Fanuc KAREL source: kt00264.KL

-- PROVISIONAL review KL for V770-1; original PC SHA256 e8cb45a23f48b17e567031bccddfba465cc350efa91dea444729adb3129dde7d
-- Incomplete behavior may be omitted. Consult companion uncertainty JSON. Do not deploy.
PROGRAM KT00264
%NOLOCKGROUP
VAR
  R1 : REAL
  OUT : BOOLEAN
-- UNRESOLVED_DECL H2 type=002017
BEGIN
  -- UNRESOLVED_PC offsets 5-16; opcodes 2E,23
  -- UNRESOLVED_PC offsets 21-35; opcodes 2E,22,9D,33,B4
  -- UNRESOLVED_PC offsets 40-63; opcodes 21,22,9D,33,B3,64,6D,23
  -- UNRESOLVED_PC offsets 68-72; opcodes 7F
END KT00264
